PROGRAM HMI
VAR
END_VAR

// if clear all faults, reset abort status
IF HMI_DB.ClearFaultPB = TRUE THEN
	Trips_DB.ChargedTimerRunout := FALSE;
	Trips_DB.ChargingTimerRunout := FALSE;
	Trips_DB.DumpTimerRunout := FALSE;
	Trips_DB.ChargerSummaryFault := FALSE;
	Trips_DB.ShortingSystemUnknown := FALSE;
END_IF

IF Trips_DB.ChargedTimerRunout = TRUE OR 
	Trips_DB.ChargingTimerRunout = TRUE //OR 
	//Trips_DB.DumpTimerRunout = TRUE 
	THEN
		Trips_DB.TimerRunOutON := TRUE; 
		ELSE
			Trips_DB.TimerRunOutON := FALSE;
		END_IF

END_PROGRAM

(* stored: Version 1.1.0.1, ProductVersion 3.1.4024.11
   POU HMI: Id {dcabf1a6-3ca3-40de-943d-43b2e4fd41d0}, SpecialFunc None *)
